// TwinCAT 3 PLC project Untitled1
// ProgramVersion: 3.1.4023.0
// libraries:
//   Tc2_Standard, * (Beckhoff Automation GmbH)
//   Tc2_System, * (Beckhoff Automation GmbH)
//   Tc3_Module, * (Beckhoff Automation GmbH)
// project tree:
//   DUTs/ DUT_oil_level.TcDUT, ST_pCraneParameters.TcDUT
//   / GlobalTextList.TcGTLO, PlcTask.TcTTO, Visualization Manager.TcVMO (not stored)
//   GVLs/ Inputs.TcGVL, Outputs.TcGVL, Parameters.TcGVL
//   POUs/ CraneSimulation.TcPOU, F_degToRad.TcPOU, MAIN.TcPOU
//   VISUs/ Visualization.TcVIS
// real-time tasks:
//   TASK PlcTask: cycle T#10ms, priority 20, ADS port 350

CONFIGURATION Untitled1
    RESOURCE PLC ON TwinCAT3
        TASK PlcTask(INTERVAL := T#10ms, PRIORITY := 20);
        PROGRAM MAIN WITH PlcTask : MAIN;
    END_RESOURCE
END_CONFIGURATION

// ---- DUTs/DUT_oil_level.TcDUT
{attribute 'qualified_only'}
{attribute 'strict'}
TYPE DUT_oil_level :
(
	VeryLow,Low,High,VeryHigh,OK
);
END_TYPE

// ---- DUTs/ST_pCraneParameters.TcDUT
TYPE ST_pCraneParameters :
STRUCT
	fCycleTime : LREAL := 10E-2;
	fInitialVelocity : REAL := 0;
	fInitialPosition : REAL := 0;
	fT1 : REAL := 0;
	fT2 : REAL := 30;
	fT3 : REAL := 60;
	fStartPos : REAL := 0;
	fMidPos : LREAL := 1;
	fEndPos : REAL := 0;
END_STRUCT
END_TYPE

// ---- GVLs/Inputs.TcGVL
{attribute 'qualified_only'}
VAR_GLOBAL
	bEnable : BOOL;
	bStart : BOOL;
	bReset : BOOL;
	fCylinderVelocityReference : REAL;
	bAutoMode : BOOL := TRUE;
	fManualCylinderPositionReference : REAL;
END_VAR

// ---- GVLs/Outputs.TcGVL
{attribute 'qualified_only'}
VAR_GLOBAL
	bSimRunning : BOOL;
	fSimulationTime : LREAL;
	fCylinderVelocity : LREAL;
	fCylinderPosition : LREAL;
END_VAR

// ---- GVLs/Parameters.TcGVL
{attribute 'qualified_only'}
VAR_GLOBAL
	pCraneParameters : ST_pCraneParameters;
	aTestArray : ARRAY[0..5] OF REAL := [0,1,2,3,4,5];
	fLowerDeadBand : LREAL := 0.1;
END_VAR

// ---- POUs/MAIN.TcPOU
PROGRAM MAIN
VAR
END_VAR


CraneSimulation();


//IF Inputs.bStart THEN
//	Outputs.bSimRunning := TRUE;
//	ELSE
//		Outputs.bSimRunning := FALSE;
//END_IF

END_PROGRAM

// ---- POUs/CraneSimulation.TcPOU
PROGRAM CraneSimulation
VAR
	fTime : LREAL;
	fOilLevelSensor : LREAL;
	eOilLevelAlarms : DUT_oil_level;
	fCraneAngle : LREAL;
	fCraneAngleDeg : LREAL;
END_VAR

IF inputs.bAutoMode AND inputs.bStart THEN
	fTime := fTime + parameters.pCraneParameters.fCycleTime;
ELSE
	fTime := 0;
END_IF

IF fTime > 0 AND inputs.bAutoMode THEN
	outputs.bSimRunning := TRUE;
END_IF
IF outputs.bSimRunning THEN
	IF fTime > 0 AND fTime <= parameters.pCraneParameters.fT2 THEN
		outputs.fCylinderVelocity := 1/(parameters.pCraneParameters.fT2);
		outputs.fCylinderPosition := outputs.fCylinderVelocity*fTime;
		parameters.pCraneParameters.fMidPos := outputs.fCylinderPosition;//saved for next loop
	ELSIF fTime > parameters.pCraneParameters.fT2 AND fTime <= parameters.pCraneParameters.fT3 THEN
		outputs.fCylinderVelocity := -1/(parameters.pCraneParameters.fT3-Parameters.pCraneParameters.fT2);
		outputs.fCylinderPosition := outputs.fCylinderVelocity*(fTime-parameters.pCraneParameters.fT2) + parameters.pCraneParameters.fMidPos;
	ELSE
		outputs.fCylinderVelocity := 0;
	END_IF

//	outputs.fCylinderVelocity := inputs.fCylinderVelocityReference;
//	outputs.fCylinderPosition := 0.5*outputs.fCylinderVelocity*fTime*fTime + parameters.fInitialVelocity*fTime + parameters.fInitialPosition;
END_IF


IF inputs.bReset THEN
	fTime := 0;
	inputs.bStart := FALSE;
	inputs.bEnable := FALSE;
	inputs.bReset := FALSE;
	outputs.fCylinderPosition := parameters.pCraneParameters.fInitialPosition;
	outputs.fCylinderVelocity := parameters.pCraneParameters.fInitialVelocity;
END_IF
//oil level
IF fOilLevelSensor < 20 THEN
	eOilLevelAlarms := DUT_oil_level.VeryLow;
	ELSIF fOilLevelSensor > 200 THEN
		eOilLevelAlarms := DUT_oil_level.VeryHigh;
	ELSE
		eOilLevelAlarms := DUT_oil_level.OK;		
END_IF
fCraneAngle := F_degToRad(fDeg := fCraneAngleDeg);

END_PROGRAM

// ---- POUs/F_degToRad.TcPOU
FUNCTION F_degToRad : LREAL
VAR_INPUT
	fDeg : LREAL;
END_VAR
VAR
	piii :LREAL := 3.14;
END_VAR

F_degToRad := fDeg*(piii/180);

END_FUNCTION

// ---- GlobalTextList.TcGTLO
TEXTLIST GlobalTextList
  253 = 'CylinderPosition: %f [m]'
  785 = 'CylinderVelocity: %f [m/s]'
  859 = 'cylinderVelocityReference: %f [m/s]'
  693 = 'CylinderVelocityReference: %f [m/s]'
  951 = 'OilLevelStatus: %i '
  776 = 'Time: %f [m]'
  535 = 'Time: %f [s]'
END_TEXTLIST

// ---- VISUs/Visualization.TcVIS
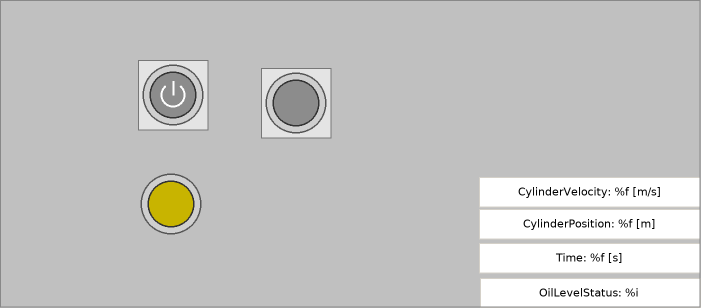
VISUALIZATION Visualization  // 701x308
    PowerSwitch (138,60 70x70), variable: Inputs.bStart, behaviour: TOGGLE, style: Switch-PowerSwitch-Gray
    Lamp1 (136,169 70x70), variable: Outputs.bSimRunning, style: Lamp-Lamp1-Yellow
    Textfield (479,177 221x30), "CylinderVelocity: %f [m/s]", text variable: Outputs.fCylinderVelocity
    Textfield (479,209 221x30), "CylinderPosition: %f [m]", text variable: Outputs.fCylinderPosition
    PushSwitch (261,68 70x70), variable: Inputs.bReset, behaviour: TOGGLE, style: Switch-PushSwitch-Gray
    Textfield (479,243 221x30), "Time: %f [s]", text variable: CraneSimulation.fTime
    Textfield (480,278 221x30), "OilLevelStatus: %i", text variable: CraneSimulation.eOilLevelAlarms
END_VISUALIZATION
